{attribute 'qualified_only'}
{attribute 'strict'}
TYPE Mode :
(
	prod 		:= 111,
	maint		:= 222
);
END_TYPE

(* stored: Version 1.1.0.1, ProductVersion 3.1.4020.12
   DUT Mode: Id {57dbb37e-5b2b-4771-af83-c584018a0eb3} *)
